PROGRAM MAIN
VAR
END_VAR

END_PROGRAM

(* stored: Version 1.1.0.1
   POU MAIN: Id {6c92053a-ac80-4506-94ff-e9aac0f40b95} *)
